FUNCTION_BLOCK MECH2_DIAGL (* Locally Coupled and Clocked Diagnostics for a Bidirectional Mechanism *)
  (* Standard: 61499-1; Classification: Diagnostics; ApplicationDomain: Mechanisms *)
  (* Version 0.2, 2005-06-01, JHC, Holobloc Inc, Recompiled with new emitter. *)
  (* Version 0.1, 2004-10-20, JHC, Rockwell Automation, Renamed to replace old MECH2_DIAG. *)
  (* Version 0.0, 2004-09-26, JHC, Rockwell Automation *)
  (* Compiler header: package fb.rt.mva; import fb.rt.net.*; *)
  (* Compiler classdef: public class MECH2_DIAGL extends FBMVCD *)
  (* Compiler Java IBM Jikes 1.06 *)
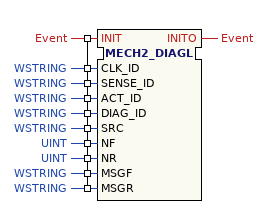
  EVENT_INPUT
    INIT WITH SENSE_ID, ACT_ID, DIAG_ID, SRC, NF, NR, MSGF, MSGR, CLK_ID;
  END_EVENT
  EVENT_OUTPUT
    INITO;
  END_EVENT
  VAR_INPUT
    CLK_ID : WSTRING := "DIAG_CLK"; (* Diagnostic Clock Local Channel ID *)
    SENSE_ID : WSTRING; (* Sensor channel ID from Model *)
    ACT_ID : WSTRING; (* Actuator channel ID from Controller *)
    DIAG_ID : WSTRING; (* Diagnostic output channel ID *)
    SRC : WSTRING; (* Diagnostic Source ID *)
    NF : UINT; (* Forward Motion Timeout Period in CLK cycles *)
    NR : UINT; (* Reverse Motion Timeout Period in CLK cycles *)
    MSGF : WSTRING := "TIMEOUT_ADVANCING"; (* Message for fault on forward motion *)
    MSGR : WSTRING := "TIMEOUT_RETRACTING"; (* Message for fault on reverse motion *)
  END_VAR
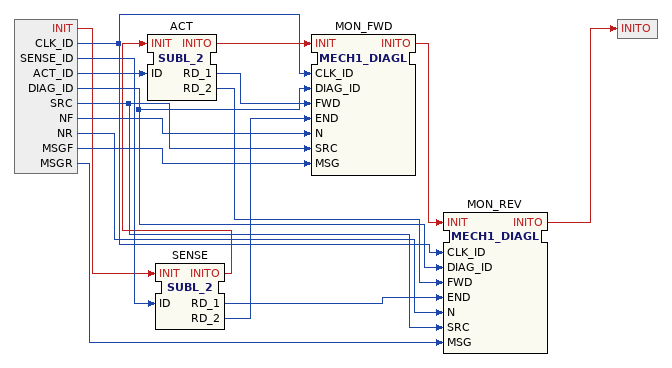
  FBS
    ACT : SUBL_2;
    SENSE : SUBL_2;
    MON_FWD : MECH1_DIAGL;
    MON_REV : MECH1_DIAGL;
  END_FBS
  EVENT_CONNECTIONS
    INIT TO SENSE.INIT;
    SENSE.INITO TO ACT.INIT;
    ACT.INITO TO MON_FWD.INIT;
    MON_FWD.INITO TO MON_REV.INIT;
    MON_REV.INITO TO INITO;
  END_CONNECTIONS
  DATA_CONNECTIONS
    ACT_ID TO ACT.ID;
    SENSE_ID TO SENSE.ID;
    CLK_ID TO MON_FWD.CLK_ID;
    DIAG_ID TO MON_FWD.DIAG_ID;
    ACT.RD_1 TO MON_FWD.FWD;
    NF TO MON_FWD.N;
    SRC TO MON_FWD.SRC;
    MSGF TO MON_FWD.MSG;
    CLK_ID TO MON_REV.CLK_ID;
    DIAG_ID TO MON_REV.DIAG_ID;
    ACT.RD_2 TO MON_REV.FWD;
    NR TO MON_REV.N;
    SRC TO MON_REV.SRC;
    MSGR TO MON_REV.MSG;
    SENSE.RD_1 TO MON_REV.END;
    SENSE.RD_2 TO MON_FWD.END;
  END_CONNECTIONS
END_FUNCTION_BLOCK
